FUNCTION_BLOCK BLINKER (* Composite Function Block Type *)
  (* Standard: 61499-2 *)
  (* Version 0.0, 1/1/2023, Dmitrii, Flexbridge AB, template *)
  PACKAGE Main;
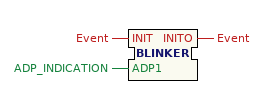
  EVENT_INPUT
    INIT; (* Initialization Request *)
  END_EVENT
  EVENT_OUTPUT
    INITO; (* Initialization Confirm *)
  END_EVENT
  SOCKETS
    ADP1 : ADP_INDICATION;
  END_SOCKETS
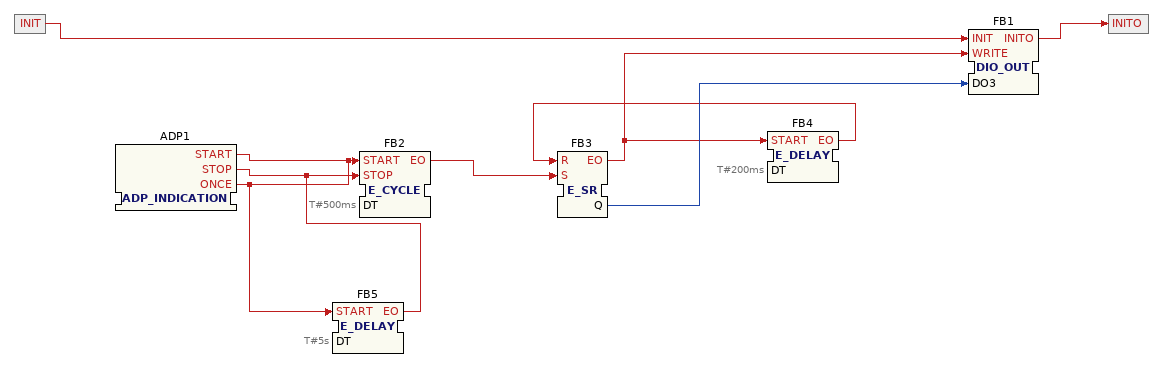
  FBS
    FB1 : DIO_OUT;
    FB2 : E_CYCLE(DT := T#500ms);
    FB3 : E_SR;
    FB4 : E_DELAY(DT := T#200ms);
    FB5 : E_DELAY(DT := T#5s);
  END_FBS
  EVENT_CONNECTIONS
    INIT TO FB1.INIT;
    FB1.INITO TO INITO;
    FB3.EO TO FB4.START;
    FB4.EO TO FB3.R;
    FB2.EO TO FB3.S;
    FB3.EO TO FB1.WRITE;
    ADP1.START TO FB2.START;
    ADP1.STOP TO FB2.STOP;
    ADP1.ONCE TO FB2.START;
    ADP1.ONCE TO FB5.START;
    FB5.EO TO FB2.STOP;
  END_CONNECTIONS
  DATA_CONNECTIONS
    FB3.Q TO FB1.DO3;
  END_CONNECTIONS
END_FUNCTION_BLOCK
